{attribute 'qualified_only'}
{attribute 'strict'}
{attribute 'to_string'}
TYPE eValvePosition :
(
	Up := 0,
	Down:=1,
	Unkown:=2
);
END_TYPE

(* stored: Version 1.1.0.1
   DUT eValvePosition: Id {de4025fc-2a36-498c-9c5b-609ad1be65e4} *)
